SUBAPPLICATION Uebung_120 (* Übung zu ISOBUS Name *)
  (* Standard: 61499-2; Description: Copyright (c) 2023 Meisterschulen am Ostbahnhof This program and the accompanying materials are made available under the terms of the Eclipse Public License 2.0 which is available at https://www.eclipse.org/legal/epl-2.0/ SPDX-License-Identifier: EPL-2.0 *)
  (* Version 1.0, 2023-10-23, Franz Höpfinger, Meisterschulen am Ostbahnhof, initial API and implementation and/or initial documentation *)
  PACKAGE Uebungen;
  IMPORT Uebungen::const::Uebung_120_129::Filter::ADD_ALL_PASS;
  IMPORT Uebungen::const::Uebung_120_129::Filter::FLT_ALL_PASS;
  IMPORT isobus::pgn::ISOUSERHOME_e::network;
  IMPORT isobus::pgn::ISO_CAN_NODE::NODE1;
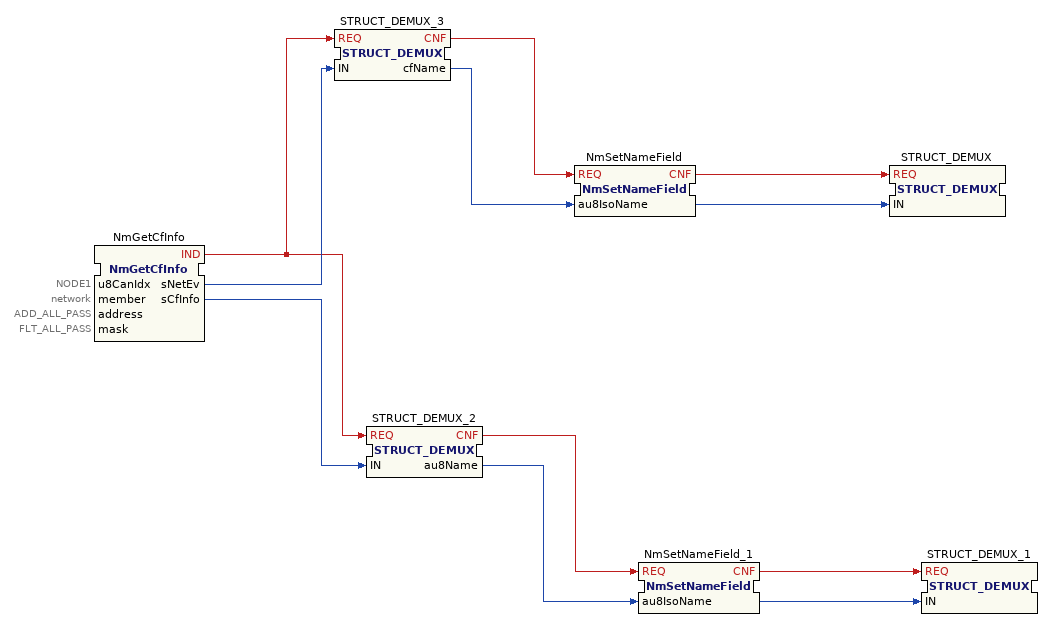
  (* mit einem Event an RSP wird der nächste ACL abgefragt. *)
  FBS
    NmGetCfInfo : isobus::pgn::NmGetCfInfo(u8CanIdx := NODE1, member := network, address := ADD_ALL_PASS, mask := FLT_ALL_PASS);
    STRUCT_DEMUX_2 : eclipse4diac::convert::STRUCT_DEMUX; {SET_ATTRIBUTE(StructuredType, isobus::pgn::CF_INFO_T)}
    STRUCT_DEMUX_3 : eclipse4diac::convert::STRUCT_DEMUX; {SET_ATTRIBUTE(StructuredType, isobus::pgn::ISONETEVENT_T)}
    NmSetNameField : isobus::pgn::NmSetNameField;
    NmSetNameField_1 : isobus::pgn::NmSetNameField;
    STRUCT_DEMUX : eclipse4diac::convert::STRUCT_DEMUX; {SET_ATTRIBUTE(StructuredType, isobus::pgn::NAMEFIELD_T)}
    STRUCT_DEMUX_1 : eclipse4diac::convert::STRUCT_DEMUX; {SET_ATTRIBUTE(StructuredType, isobus::pgn::NAMEFIELD_T)}
  END_FBS
  EVENT_CONNECTIONS
    NmGetCfInfo.IND TO STRUCT_DEMUX_3.REQ;
    NmGetCfInfo.IND TO STRUCT_DEMUX_2.REQ;
    STRUCT_DEMUX_3.CNF TO NmSetNameField.REQ;
    STRUCT_DEMUX_2.CNF TO NmSetNameField_1.REQ;
    NmSetNameField.CNF TO STRUCT_DEMUX.REQ;
    NmSetNameField_1.CNF TO STRUCT_DEMUX_1.REQ;
  END_CONNECTIONS
  DATA_CONNECTIONS
    NmGetCfInfo.sNetEv TO STRUCT_DEMUX_3.IN;
    NmGetCfInfo.sCfInfo TO STRUCT_DEMUX_2.IN;
    STRUCT_DEMUX_3.cfName TO NmSetNameField.au8IsoName;
    STRUCT_DEMUX_2.au8Name TO NmSetNameField_1.au8IsoName;
    NmSetNameField. TO STRUCT_DEMUX.IN;
    NmSetNameField_1. TO STRUCT_DEMUX_1.IN;
  END_CONNECTIONS
END_SUBAPPLICATION
